(* Step MesCheckResult_1 *)
(* EN: Step structure *)
IF Step_MesCheckResult_1_active THEN
  (* Timeout Check *)
  IF (SYS_TIME - Step_MesCheckResult_1_entry_time) > MesCheckResult_1.T_MAX THEN Step_MesCheckResult_1_timeout := TRUE; END_IF;

  IF Action_MesCheckResult_1_Exec THEN
    "PLCtoMES"."PLC.Unload_Station7DataSaveReq" := TRUE;
    Action_MesCheckResult_1_Done := TRUE;
  END_IF;
END_IF;

(* Step Bypass_1 *)
(* EN: Step structure *)
IF Step_Bypass_1_active THEN
  (* Timeout Check *)
  IF (SYS_TIME - Step_Bypass_1_entry_time) > Bypass_1.T_MAX THEN Step_Bypass_1_timeout := TRUE; END_IF;

  IF Action_Bypass_1_Exec THEN
    Action_Bypass_1_Done := TRUE;
  END_IF;
END_IF;

(* Step ResetMesUnloadRequest_1 *)
(* EN: Step structure *)
IF Step_ResetMesUnloadRequest_1_active THEN
  (* Timeout Check *)
  IF (SYS_TIME - Step_ResetMesUnloadRequest_1_entry_time) > ResetMesUnloadRequest_1.T_MAX THEN Step_ResetMesUnloadRequest_1_timeout := TRUE; END_IF;

  IF Action_ResetMesUnloadRequest_1_Exec THEN
    "PLCtoMES"."PLC.Unload_Station7DataSaveReq" := FALSE;
    "MEStoPLC"."MES.Unload_ResultsStored7OK" := FALSE;
    "MEStoPLC"."MES.Unload_ResultsStored7NG" := FALSE;
    "MEStoPLC"."MES.Unload_ResultsStored7ReqMesDone" := FALSE;
    Action_ResetMesUnloadRequest_1_Done := TRUE;
  END_IF;
END_IF;

(* Step Step314 *)
(* EN: Step structure *)
IF Step_Step314_active THEN
  (* Timeout Check *)
  IF (SYS_TIME - Step_Step314_entry_time) > Step314.T_MAX THEN Step_Step314_timeout := TRUE; END_IF;

  IF Action_Step314_Exec THEN
    Action_Step314_Done := TRUE;
  END_IF;
END_IF;

(* Step MESOverTime *)
(* EN: Step structure *)
IF Step_MESOverTime_active THEN
  (* Timeout Check *)
  IF (SYS_TIME - Step_MESOverTime_entry_time) > MESOverTime.T_MAX THEN Step_MESOverTime_timeout := TRUE; END_IF;

  IF Action_MESOverTime_Exec THEN
    "ST10_DeviceError".MES_Error.CheckInResultOverTime_7 := TRUE;
    Action_MESOverTime_Done := TRUE;
  END_IF;
END_IF;

(* Step ok_1 *)
(* EN: Step structure *)
IF Step_Ok_1_active THEN
  (* Timeout Check *)
  IF (SYS_TIME - Step_Ok_1_entry_time) > Ok_1.T_MAX THEN Step_Ok_1_timeout := TRUE; END_IF;

  IF Action_Ok_1_Exec THEN
    IF "AutoProcessData".B_Press2.PartStatus = 480 THEN
      "AutoProcessData".B_Press2.PartStatus := 499;
    END_IF;
    Action_Ok_1_Done := TRUE;
  END_IF;
END_IF;

(* Step Prepare MES CheckData_1 *)
(* EN: Step structure *)
IF Step_PrepareMESCheckData_1_active THEN
  (* Timeout Check *)
  IF (SYS_TIME - Step_PrepareMESCheckData_1_entry_time) > PrepareMESCheckData_1.T_MAX THEN Step_PrepareMESCheckData_1_timeout := TRUE; END_IF;

  IF Action_PrepareMESCheckData_1_Exec THEN
    Action_PrepareMESCheckData_1_Done := TRUE;
  END_IF;
END_IF;

(* Transition 399: MES Result OK_1 -> MES Check Finish *)
IF Step_MESResultOK_1_active AND ( "AutoProcessData".B_Press2.PartStatus = 499 ) THEN
  Step_MESResultOK_1_active := FALSE;
  Action_MESResultOK_1_Exec := FALSE;

  Step_MESCheckFinish_active := TRUE;
  Step_MESCheckFinish_entry_time := SYS_TIME; (* Reset Timer *)
  Action_MESCheckFinish_Exec := TRUE;

  Trans_Trans321_executed := TRUE;
END_IF;

(* Transition 500: MES Result -> Bypass_1 *)
IF Step_MESResult_active AND ( TRUE ) THEN
  Step_MESResult_active := FALSE;
  Action_MESResult_Exec := FALSE;

  Step_Bypass_1_active := TRUE;
  Step_Bypass_1_entry_time := SYS_TIME; (* Reset Timer *)
  Action_Bypass_1_Exec := TRUE;

  Trans_Trans407_executed := TRUE;
END_IF;

(* Transition 515: MES Check Finish -> RobotPick (Jump) *)
IF Step_MESCheckFinish_active AND ( TRUE ) THEN
  Step_MESCheckFinish_active := FALSE;
  Action_MESCheckFinish_Exec := FALSE;

  Step_RobotPick_active := TRUE;
  Step_RobotPick_entry_time := SYS_TIME; (* Reset Timer *)
  Action_RobotPick_Exec := TRUE;

  Trans_Trans619_executed := TRUE;
END_IF;

(* Transition 308: Prepare MES CheckData_1 -> MesCheckResult_1 *)
IF Step_PrepareMESCheckData_1_active AND ( PrepareMESCheckData_1.T > T#300ms ) THEN
  Step_PrepareMESCheckData_1_active := FALSE;
  Action_PrepareMESCheckData_1_Exec := FALSE;

  Step_MesCheckResult_1_active := TRUE;
  Step_MesCheckResult_1_entry_time := SYS_TIME; (* Reset Timer *)
  Action_MesCheckResult_1_Exec := TRUE;

  Trans_Trans16_executed := TRUE;
END_IF;

(* Transition 315: MesCheckResult_1 -> MESResultOK_1 *)
IF Step_MesCheckResult_1_active AND ( (NOT "MEStoPLC"."MES.Unload_ResultsStored7OK") AND "MEStoPLC"."MES.Unload_ResultsStored7NG" AND "MEStoPLC"."MES.Unload_ResultsStored7ReqMesDone" ) THEN
  Step_MesCheckResult_1_active := FALSE;
  Action_MesCheckResult_1_Exec := FALSE;

  Step_MESResultOK_1_active := TRUE;
  Step_MESResultOK_1_entry_time := SYS_TIME; (* Reset Timer *)
  Action_MESResultOK_1_Exec := TRUE;

  Trans_Trans315_executed := TRUE;
END_IF;

(* Transition 321: Step313 -> CheckFinish_1 *)
IF Step_Step313_active AND ( TRUE ) THEN
  Step_Step313_active := FALSE;
  Action_Step313_Exec := FALSE;

  Step_CheckFinish_1_active := TRUE;
  Step_CheckFinish_1_entry_time := SYS_TIME; (* Reset Timer *)
  Action_CheckFinish_1_Exec := TRUE;

  Trans_Trans319_executed := TRUE; (* Original: Trans321. Typo in XML? *)
END_IF;

(* Transition 322: MesCheckResult_1 -> MESCheckNG_3 *)
IF Step_MesCheckResult_1_active AND ( "AutoProcessData".B_Press2.PartStatus = 452 ) THEN
  Step_MesCheckResult_1_active := FALSE;
  Action_MesCheckResult_1_Exec := FALSE;

  Step_MESCheckNG_3_active := TRUE;
  Step_MESCheckNG_3_entry_time := SYS_TIME; (* Reset Timer *)
  Action_MESCheckNG_3_Exec := TRUE;

  Trans_Trans322_executed := TRUE;
END_IF;

(* Transition 323: MESCheckNG_3 -> MES Result OK_1 *)
IF Step_MESCheckNG_3_active AND ( "MEStoPLC"."MES.Unload_ResultsStored7OK" AND (NOT "MEStoPLC"."MES.Unload_ResultsStored7NG") AND "MEStoPLC"."MES.Unload_ResultsStored7ReqMesDone" AND ("AutoProcessData".B_Press2.PartStatus <> 450) AND ("AutoProcessData".B_Press2.PartStatus <> 455) ) THEN
  Step_MESCheckNG_3_active := FALSE;
  Action_MESCheckNG_3_Exec := FALSE;

  Step_MESResultOK_1_active := TRUE;
  Step_MESResultOK_1_entry_time := SYS_TIME; (* Reset Timer *)
  Action_MESResultOK_1_Exec := TRUE;

  Trans_Trans323_executed := TRUE;
END_IF;

(* Transition 324: MESCheckNG_3 -> Step314 *)
IF Step_MESCheckNG_3_active AND ( (NOT "MEStoPLC"."MES.Load_Station7ReqMesDone") AND (MesCheckResult_1.T > T#10s) ) THEN
  Step_MESCheckNG_3_active := FALSE;
  Action_MESCheckNG_3_Exec := FALSE;

  Step_Step314_active := TRUE;
  Step_Step314_entry_time := SYS_TIME; (* Reset Timer *)
  Action_Step314_Exec := TRUE;

  Trans_Trans324_executed := TRUE;
END_IF;

(* Transition 325: Bypass_1 -> ResetMesUnloadRequest_1 *)
IF Step_Bypass_1_active AND ( (NOT "Station_Sys".Cmd.OnOffLine) ) THEN
  Step_Bypass_1_active := FALSE;
  Action_Bypass_1_Exec := FALSE;

  Step_ResetMesUnloadRequest_1_active := TRUE;
  Step_ResetMesUnloadRequest_1_entry_time := SYS_TIME; (* Reset Timer *)
  Action_ResetMesUnloadRequest_1_Exec := TRUE;

  Trans_Online_1_executed := TRUE; (* Original: Trans325. Typo in XML? *)
END_IF;

(* Transition 326: ResetMesUnloadRequest_1 -> Prepare MES CheckData_1 *)
IF Step_ResetMesUnloadRequest_1_active AND ( NOT "PLCtoMES"."PLC.Unload_Station7DataSaveReq" AND NOT "MEStoPLC"."MES.Unload_ResultsStored7OK" AND NOT "MEStoPLC"."MES.Unload_ResultsStored7NG" AND NOT "MEStoPLC"."MES.Unload_ResultsStored7ReqMesDone" ) THEN
  Step_ResetMesUnloadRequest_1_active := FALSE;
  Action_ResetMesUnloadRequest_1_Exec := FALSE;

  Step_PrepareMESCheckData_1_active := TRUE;
  Step_PrepareMESCheckData_1_entry_time := SYS_TIME; (* Reset Timer *)
  Action_PrepareMESCheckData_1_Exec := TRUE;

  Trans_Trans260_executed := TRUE;
END_IF;

(* Transition 327: Bypass_1 -> ok_1 *)
IF Step_Bypass_1_active AND ( "Station_Sys".Cmd.OnOffLine ) THEN
  Step_Bypass_1_active := FALSE;
  Action_Bypass_1_Exec := FALSE;

  Step_Ok_1_active := TRUE;
  Step_Ok_1_entry_time := SYS_TIME; (* Reset Timer *)
  Action_Ok_1_Exec := TRUE;

  Trans_Trans327_executed := TRUE;
END_IF;

(* Transition 328: MESOverTime -> Bypass_1 (Jump) *)
IF Step_MESOverTime_active AND ( TRUE ) THEN
  Step_MESOverTime_active := FALSE;
  Action_MESOverTime_Exec := FALSE;

  Step_Bypass_1_active := TRUE;
  Step_Bypass_1_entry_time := SYS_TIME; (* Reset Timer *)
  Action_Bypass_1_Exec := TRUE;

  Trans_Trans329_executed := TRUE; (* Original: Trans328. Typo in XML? *)
END_IF;

(* Transition 331: ok_1 -> Step314 *)
IF Step_Ok_1_active AND ( TRUE ) THEN
  Step_Ok_1_active := FALSE;
  Action_Ok_1_Exec := FALSE;

  Step_Step314_active := TRUE;
  Step_Step314_entry_time := SYS_TIME; (* Reset Timer *)
  Action_Step314_Exec := TRUE;

  Trans_Trans328_executed := TRUE; (* Original: Trans331. Typo in XML? *)
END_IF;

(* Transition 330: Step314 -> MESOverTime *)
IF Step_Step314_active AND ( TRUE ) THEN
  Step_Step314_active := FALSE;
  Action_Step314_Exec := FALSE;

  Step_MESOverTime_active := TRUE;
  Step_MESOverTime_entry_time := SYS_TIME; (* Reset Timer *)
  Action_MESOverTime_Exec := TRUE;

  Trans_Trans327_executed := TRUE; (* Original: Trans330. Typo in XML? *)
END_IF;


(* Sequence: S600-S699 RobotPick *)
(* S600-S699工件放行 *)
(* Step RobotPick *)
(* EN: Step structure *)
IF Step_RobotPick_active THEN
  (* Timeout Check *)
  IF (SYS_TIME - Step_RobotPick_entry_time) > RobotPick.T_MAX THEN Step_RobotPick_timeout := TRUE; END_IF;

  IF Action_RobotPick_Exec THEN
    Action_RobotPick_Done := TRUE;
  END_IF;
END_IF;

(* Step ProcessFinsh *)
(* ZH-CN: 正式使用时，需要激活复位空循环 *)
(* EN: Step structure *)
IF Step_ProcessFinsh_3_active THEN
  (* Timeout Check *)
  IF (SYS_TIME - Step_ProcessFinsh_3_entry_time) > ProcessFinsh_3.T_MAX THEN Step_ProcessFinsh_3_timeout := TRUE; END_IF;

  IF Action_ProcessFinsh_3_Exec THEN
    #ioPM_Inface.ProcessComplete := TRUE;
    #ioPM_Inface.ProcessStart := FALSE;
    Action_ProcessFinsh_3_Done := TRUE;
  END_IF;
END_IF;

(* Step DataClear *)
(* EN: Step structure *)
IF Step_DataClear_active THEN
  (* Timeout Check *)
  IF (SYS_TIME - Step_DataClear_entry_time) > DataClear.T_MAX THEN Step_DataClear_timeout := TRUE; END_IF;

  IF Action_DataClear_Exec THEN
    #ioPM_Inface.ProcessResult := 0;
    #ioStatus := 0;
    Action_DataClear_Done := TRUE;
  END_IF;
END_IF;

(* Step Request robot pick *)
(* EN: Step structure *)
IF Step_RequestRobotPick_active THEN
  (* Timeout Check *)
  IF (SYS_TIME - Step_RequestRobotPick_entry_time) > RequestRobotPick.T_MAX THEN Step_RequestRobotPick_timeout := TRUE; END_IF;

  IF Action_RequestRobotPick_Exec THEN
    "AutoProcessControl".B_Press_2.Robot3PickPrimit := TRUE;
    Action_RequestRobotPick_Done := TRUE;
  END_IF;
END_IF;

(* Step Wait robot finish task *)
(* EN: Step structure *)
IF Step_WaitRobotFinishTask_1_active THEN
  (* Timeout Check *)
  IF (SYS_TIME - Step_WaitRobotFinishTask_1_entry_time) > WaitRobotFinishTask_1.T_MAX THEN Step_WaitRobotFinishTask_1_timeout := TRUE; END_IF;

  IF Action_WaitRobotFinishTask_1_Exec THEN
    Action_WaitRobotFinishTask_1_Done := TRUE;
  END_IF;
END_IF;

(* Step DataMove *)
(* EN: Step structure *)
IF Step_DataMove_active THEN
  (* Timeout Check *)
  IF (SYS_TIME - Step_DataMove_entry_time) > DataMove.T_MAX THEN Step_DataMove_timeout := TRUE; END_IF;

  IF Action_DataMove_Exec THEN
    Action_DataMove_Done := TRUE;
  END_IF;
END_IF;

(* Step Wait robot in safety area *)
(* EN: Step structure *)
IF Step_WaitRobotInSafetyArea_active THEN
  (* Timeout Check *)
  IF (SYS_TIME - Step_WaitRobotInSafetyArea_entry_time) > WaitRobotInSafetyArea.T_MAX THEN Step_WaitRobotInSafetyArea_timeout := TRUE; END_IF;

  IF Action_WaitRobotInSafetyArea_Exec THEN
    Action_WaitRobotInSafetyArea_Done := TRUE;
  END_IF;
END_IF;

(* Step PressProgram_1 *)
(* EN: Step structure *)
IF Step_PressProgram_1_active THEN
  (* Timeout Check *)
  IF (SYS_TIME - Step_PressProgram_1_entry_time) > PressProgram_1.T_MAX THEN Step_PressProgram_1_timeout := TRUE; END_IF;

  IF Action_PressProgram_1_Exec THEN
    IF NOT "ST10_GeneralData".FunctionDeSelect.B.FunctionDeSelected_TestPress375A1 THEN
      "DB_maXYmosNC2".ProgNo := 1;
    END_IF;
    Action_PressProgram_1_Done := TRUE;
  END_IF;
END_IF;

(* Step PressHoming_1 *)
(* EN: Step structure *)
IF Step_PressHoming_1_active THEN
  (* Timeout Check *)
  IF (SYS_TIME - Step_PressHoming_1_entry_time) > PressHoming_1.T_MAX THEN Step_PressHoming_1_timeout := TRUE; END_IF;

  IF Action_PressHoming_1_Exec THEN
    "DB_maXYmosNC2".Homing := TRUE;
    Action_PressHoming_1_Done := TRUE;
  END_IF;
END_IF;

(* Step PressReady?_1 *)
(* EN: Step structure *)
IF Step_PressReady_q_1_active THEN
  (* Timeout Check *)
  IF (SYS_TIME - Step_PressReady_q_1_entry_time) > PressReady_q_1.T_MAX THEN Step_PressReady_q_1_timeout := TRUE; END_IF;

  IF Action_PressReady_q_1_Exec THEN
    Action_PressReady_q_1_Done := TRUE;
  END_IF;
END_IF;

(* Step PressHoming?_1 *)
(* EN: Step structure *)
IF Step_PressHoming_q_1_active THEN
  (* Timeout Check *)
  IF (SYS_TIME - Step_PressHoming_q_1_entry_time) > PressHoming_q_1.T_MAX THEN Step_PressHoming_q_1_timeout := TRUE; END_IF;

  IF Action_PressHoming_q_1_Exec THEN
    Action_PressHoming_q_1_Done := TRUE;
  END_IF;
END_IF;

(* Step Step15 *)
(* EN: Step structure *)
IF Step_Step15_active THEN
  (* Timeout Check *)
  IF (SYS_TIME - Step_Step15_entry_time) > Step15.T_MAX THEN Step_Step15_timeout := TRUE; END_IF;

  IF Action_Step15_Exec THEN
    Action_Step15_Done := TRUE;
  END_IF;
END_IF;

(* Step B-PressFitting-01CylinderToHP_1 *)
(* EN: Step structure *)
IF Step_B_PressFitting_01CylinderToHP_1_active THEN
  (* Timeout Check *)
  IF (SYS_TIME - Step_B_PressFitting_01CylinderToHP_1_entry_time) > B_PressFitting_01CylinderToHP_1.T_MAX THEN Step_B_PressFitting_01CylinderToHP_1_timeout := TRUE; END_IF;

  IF Action_B_PressFitting_01CylinderToHP_1_Exec THEN
    "ST10Cylinder".Cy[8].Inout.AutoGoHome := TRUE;
    "ST10Cylinder".Cy[8].Inout.AutoGoWork := FALSE;
    Action_B_PressFitting_01CylinderToHP_1_Done := TRUE;
  END_IF;
END_IF;

(* Transition 600: RobotPick -> PressProgram_1 *)
IF Step_RobotPick_active AND ( TRUE ) THEN
  Step_RobotPick_active := FALSE;
  Action_RobotPick_Exec := FALSE;

  Step_PressProgram_1_active := TRUE;
  Step_PressProgram_1_entry_time := SYS_TIME; (* Reset Timer *)
  Action_PressProgram_1_Exec := TRUE;

  Trans_Trans600_executed := TRUE;
END_IF;

(* Transition 604: DataClear -> ProcessFinsh *)
IF Step_DataClear_active AND ( TRUE ) THEN
  Step_DataClear_active := FALSE;
  Action_DataClear_Exec := FALSE;

  Step_ProcessFinsh_3_active := TRUE;
  Step_ProcessFinsh_3_entry_time := SYS_TIME; (* Reset Timer *)
  Action_ProcessFinsh_3_Exec := TRUE;

  Trans_Trans290_executed := TRUE;
END_IF;

(* Transition 605: ProcessFinsh -> ProcessStart (Jump) *)
IF Step_ProcessFinsh_3_active AND ( TRUE ) THEN
  Step_ProcessFinsh_3_active := FALSE;
  Action_ProcessFinsh_3_Exec := FALSE;

  Step_ProcessStart_active := TRUE;
  Step_ProcessStart_entry_time := SYS_TIME; (* Reset Timer *)
  Action_ProcessStart_Exec := TRUE;

  Trans_Trans699_executed := TRUE;
END_IF;

(* Transition 410: Request robot pick -> Wait robot finish task *)
IF Step_RequestRobotPick_active AND ( "KukaRobot3_CtrlDB".sROBtoPLC.User.Cycle.DO281_PressPickInside AND (NOT "KukaRobot3_CtrlDB".sROBtoPLC.User.Cycle.DO282_PressPickFinish) ) THEN
  Step_RequestRobotPick_active := FALSE;
  Action_RequestRobotPick_Exec := FALSE;

  Step_WaitRobotFinishTask_1_active := TRUE;
  Step_WaitRobotFinishTask_1_entry_time := SYS_TIME; (* Reset Timer *)
  Action_WaitRobotFinishTask_1_Exec := TRUE;

  Trans_Trans412_executed := TRUE;
END_IF;

(* Transition 256: Wait robot finish task -> DataMove *)
IF Step_WaitRobotFinishTask_1_active AND ( "KukaRobot3_CtrlDB".sROBtoPLC.User.Cycle.DO282_PressPickFinish ) THEN
  Step_WaitRobotFinishTask_1_active := FALSE;
  Action_WaitRobotFinishTask_1_Exec := FALSE;

  Step_DataMove_active := TRUE;
  Step_DataMove_entry_time := SYS_TIME; (* Reset Timer *)
  Action_DataMove_Exec := TRUE;

  Trans_Trans257_executed := TRUE;
END_IF;

(* Transition 257: DataMove -> Wait robot in safety area *)
IF Step_DataMove_active AND ( TRUE ) THEN
  Step_DataMove_active := FALSE;
  Action_DataMove_Exec := FALSE;

  Step_WaitRobotInSafetyArea_active := TRUE;
  Step_WaitRobotInSafetyArea_entry_time := SYS_TIME; (* Reset Timer *)
  Action_WaitRobotInSafetyArea_Exec := TRUE;

  Trans_Trans258_executed := TRUE;
END_IF;

(* Transition 258: Wait robot in safety area -> DataClear *)
IF Step_WaitRobotInSafetyArea_active AND ( "KukaRobot3_CtrlDB".sROBtoPLC.User.Home.DO177_PressPut1Area AND "KukaRobot3_CtrlDB".sROBtoPLC.User.Home.DO178_Robot2Area ) THEN
  Step_WaitRobotInSafetyArea_active := FALSE;
  Action_WaitRobotInSafetyArea_Exec := FALSE;

  Step_DataClear_active := TRUE;
  Step_DataClear_entry_time := SYS_TIME; (* Reset Timer *)
  Action_DataClear_Exec := TRUE;

  Trans_Trans261_executed := TRUE;
END_IF;

(* Transition 26: PressHoming_1 -> Step15 *)
IF Step_PressHoming_1_active AND ( "DB_maXYmosNC2".oInHomePos ) THEN
  Step_PressHoming_1_active := FALSE;
  Action_PressHoming_1_Exec := FALSE;

  Step_Step15_active := TRUE;
  Step_Step15_entry_time := SYS_TIME; (* Reset Timer *)
  Action_Step15_Exec := TRUE;

  Trans_Trans9_executed := TRUE; (* Original: Trans26. Typo in XML? *)
END_IF;

(* Transition 27: PressProgram_1 -> PressReady?_1 *)
IF Step_PressProgram_1_active AND ( TRUE ) THEN
  Step_PressProgram_1_active := FALSE;
  Action_PressProgram_1_Exec := FALSE;

  Step_PressReady_q_1_active := TRUE;
  Step_PressReady_q_1_entry_time := SYS_TIME; (* Reset Timer *)
  Action_PressReady_q_1_Exec := TRUE;

  Trans_Trans31_executed := TRUE; (* Original: Trans27. Typo in XML? *)
END_IF;

(* Transition 28: PressReady?_1 -> PressHoming?_1 *)
IF Step_PressReady_q_1_active AND ( "DB_maXYmosNC2".oReady AND "DB_maXYmosNC2".oRdyAmp ) THEN
  Step_PressReady_q_1_active := FALSE;
  Action_PressReady_q_1_Exec := FALSE;

  Step_PressHoming_q_1_active := TRUE;
  Step_PressHoming_q_1_entry_time := SYS_TIME; (* Reset Timer *)
  Action_PressHoming_q_1_Exec := TRUE;

  Trans_Trans32_executed := TRUE; (* Original: Trans28. Typo in XML? *)
END_IF;

(* Transition 29: PressHoming?_1 -> PressHoming_1 *)
IF Step_PressHoming_q_1_active AND ( NOT "DB_maXYmosNC2".oInHomePos ) THEN
  Step_PressHoming_q_1_active := FALSE;
  Action_PressHoming_q_1_Exec := FALSE;

  Step_PressHoming_1_active := TRUE;
  Step_PressHoming_1_entry_time := SYS_TIME; (* Reset Timer *)
  Action_PressHoming_1_Exec := TRUE;

  Trans_Trans33_executed := TRUE; (* Original: Trans29. Typo in XML? *)
END_IF;

(* Transition 30: PressHoming?_1 -> Step15 *)
IF Step_PressHoming_q_1_active AND ( "DB_maXYmosNC2".oInHomePos ) THEN
  Step_PressHoming_q_1_active := FALSE;
  Action_PressHoming_q_1_Exec := FALSE;

  Step_Step15_active := TRUE;
  Step_Step15_entry_time := SYS_TIME; (* Reset Timer *)
  Action_Step15_Exec := TRUE;

  Trans_Trans34_executed := TRUE; (* Original: Trans30. Typo in XML? *)
END_IF;

(* Transition 31: Step15 -> B-PressFitting-01CylinderToHP_1 *)
IF Step_Step15_active AND ( TRUE ) THEN
  Step_Step15_active := FALSE;
  Action_Step15_Exec := FALSE;

  Step_B_PressFitting_01CylinderToHP_1_active := TRUE;
  Step_B_PressFitting_01CylinderToHP_1_entry_time := SYS_TIME; (* Reset Timer *)
  Action_B_PressFitting_01CylinderToHP_1_Exec := TRUE;

  Trans_Trans35_executed := TRUE; (* Original: Trans31. Typo in XML? *)
END_IF;

(* Transition 131: B-PressFitting-01CylinderToHP_1 -> Request robot pick *)
IF Step_B_PressFitting_01CylinderToHP_1_active AND ( (NOT "ST10Cylinder".Cy[8].In.WorkPositionSensor) AND "ST10Cylinder".Cy[8].In.HomePositionSensor ) THEN
  Step_B_PressFitting_01CylinderToHP_1_active := FALSE;
  Action_B_PressFitting_01CylinderToHP_1_Exec := FALSE;

  Step_RequestRobotPick_active := TRUE;
  Step_RequestRobotPick_entry_time := SYS_TIME; (* Reset Timer *)
  Action_RequestRobotPick_Exec := TRUE;

  Trans_Trans768_executed := TRUE;
END_IF;

(* Initial Step *)
IF "RT_DATA".MOP.INIT THEN
  Step_F14_Initial_active := TRUE;
  Step_F14_Initial_entry_time := SYS_TIME;
  Action_F14_Initial_Exec := TRUE;
ELSE
  IF NOT Step_F14_Initial_active THEN
    (* Check for all transitions, and activate the next step if condition met *)
    (* Sequence S01-S99 Initial *)
    IF Step_F14_Initial_active AND Trans_Trans1_executed THEN
      Step_F14_Initial_active := FALSE;
      Action_F14_Initial_Exec := FALSE;

      Step_S2_active := TRUE;
      Step_S2_entry_time := SYS_TIME;
      Action_S2_Exec := TRUE;
    ELSIF Step_S2_active AND Trans_Trans2_executed THEN
      Step_S2_active := FALSE;
      Action_S2_Exec := FALSE;

      Step_S3_active := TRUE;
      Step_S3_entry_time := SYS_TIME;
      Action_S3_Exec := TRUE;
    ELSIF Step_S3_active AND Trans_Trans613_executed THEN
      Step_S3_active := FALSE;
      Action_S3_Exec := FALSE;

      Step_S4_active := TRUE;
      Step_S4_entry_time := SYS_TIME;
      Action_S4_Exec := TRUE;
    ELSIF Step_S4_active AND Trans_Trans3_executed THEN
      Step_S4_active := FALSE;
      Action_S4_Exec := FALSE;

      Step_S5_MESInitial_active := TRUE;
      Step_S5_MESInitial_entry_time := SYS_TIME;
      Action_S5_MESInitial_Exec := TRUE;
    ELSIF Step_S5_MESInitial_active AND Trans_Trans325_executed THEN
      Step_S5_MESInitial_active := FALSE;
      Action_S5_MESInitial_Exec := FALSE;

      Step_CheckPressGripStatus_active := TRUE;
      Step_CheckPressGripStatus_entry_time := SYS_TIME;
      Action_CheckPressGripStatus_Exec := TRUE;
    ELSIF Step_CheckPressGripStatus_active AND Trans_Trans19_executed THEN
      Step_CheckPressGripStatus_active := FALSE;
      Action_CheckPressGripStatus_Exec := FALSE;

      Step_CheckRingExist_active := TRUE;
      Step_CheckRingExist_entry_time := SYS_TIME;
      Action_CheckRingExist_Exec := TRUE;
    ELSIF Step_CheckPressGripStatus_active AND Trans_Trans20_executed THEN
      Step_CheckPressGripStatus_active := FALSE;
      Action_CheckPressGripStatus_Exec := FALSE;

      Step_B_PressFitting_01GripperCylinderToWP_active := TRUE;
      Step_B_PressFitting_01GripperCylinderToWP_entry_time := SYS_TIME;
      Action_B_PressFitting_01GripperCylinderToWP_Exec := TRUE;
    ELSIF Step_CheckPressGripStatus_active AND Trans_Trans119_executed THEN
      Step_CheckPressGripStatus_active := FALSE;
      Action_CheckPressGripStatus_Exec := FALSE;

      Step_StatusAlarm_active := TRUE;
      Step_StatusAlarm_entry_time := SYS_TIME;
      Action_StatusAlarm_Exec := TRUE;
    ELSIF Step_StatusAlarm_active AND Trans_Trans120_executed THEN
      Step_StatusAlarm_active := FALSE;
      Action_StatusAlarm_Exec := FALSE;

      Step_CheckPressGripStatus_active := TRUE;
      Step_CheckPressGripStatus_entry_time := SYS_TIME;
      Action_CheckPressGripStatus_Exec := TRUE;
    ELSIF Step_CheckRingExist_active AND Trans_Trans117_executed THEN
      Step_CheckRingExist_active := FALSE;
      Action_CheckRingExist_Exec := FALSE;

      Step_B_PressFitting_01GripperCylinderToHP_active := TRUE;
      Step_B_PressFitting_01GripperCylinderToHP_entry_time := SYS_TIME;
      Action_B_PressFitting_01GripperCylinderToHP_Exec := TRUE;
    ELSIF Step_B_PressFitting_01GripperCylinderToHP_active AND Trans_Trans765_executed THEN
      Step_B_PressFitting_01GripperCylinderToHP_active := FALSE;
      Action_B_PressFitting_01GripperCylinderToHP_Exec := FALSE;

      Step_PressProgram_active := TRUE;
      Step_PressProgram_entry_time := SYS_TIME;
      Action_PressProgram_Exec := TRUE;
    ELSIF Step_B_PressFitting_01GripperCylinderToWP_active AND Trans_Trans766_executed THEN
      Step_B_PressFitting_01GripperCylinderToWP_active := FALSE;
      Action_B_PressFitting_01GripperCylinderToWP_Exec := FALSE;

      Step_PressProgram_active := TRUE;
      Step_PressProgram_entry_time := SYS_TIME;
      Action_PressProgram_Exec := TRUE;
    ELSIF Step_PressProgram_active AND Trans_Trans10_executed THEN
      Step_PressProgram_active := FALSE;
      Action_PressProgram_Exec := FALSE;

      Step_PressReady_q_active := TRUE;
      Step_PressReady_q_entry_time := SYS_TIME;
      Action_PressReady_q_Exec := TRUE;
    ELSIF Step_PressReady_q_active AND Trans_Trans12_executed THEN
      Step_PressReady_q_active := FALSE;
      Action_PressReady_q_Exec := FALSE;

      Step_PressHoming_q_active := TRUE;
      Step_PressHoming_q_entry_time := SYS_TIME;
      Action_PressHoming_q_Exec := TRUE;
    ELSIF Step_PressHoming_q_active AND Trans_Trans15_executed THEN
      Step_PressHoming_q_active := FALSE;
      Action_PressHoming_q_Exec := FALSE;

      Step_PressHoming_active := TRUE;
      Step_PressHoming_entry_time := SYS_TIME;
      Action_PressHoming_Exec := TRUE;
    ELSIF Step_PressHoming_q_active AND Trans_Trans17_executed THEN
      Step_PressHoming_q_active := FALSE;
      Action_PressHoming_q_Exec := FALSE;

      Step_Step14_active := TRUE;
      Step_Step14_entry_time := SYS_TIME;
      Action_Step14_Exec := TRUE;
    ELSIF Step_PressHoming_active AND Trans_Trans7_executed THEN
      Step_PressHoming_active := FALSE;
      Action_PressHoming_Exec := FALSE;

      Step_Step14_active := TRUE;
      Step_Step14_entry_time := SYS_TIME;
      Action_Step14_Exec := TRUE;
    ELSIF Step_Step14_active AND Trans_Trans18_executed THEN
      Step_Step14_active := FALSE;
      Action_Step14_Exec := FALSE;

      Step_B_PressFitting_01CylinderToHP_active := TRUE;
      Step_B_PressFitting_01CylinderToHP_entry_time := SYS_TIME;
      Action_B_PressFitting_01CylinderToHP_Exec := TRUE;
    ELSIF Step_B_PressFitting_01CylinderToHP_active AND Trans_Trans767_executed THEN
      Step_B_PressFitting_01CylinderToHP_active := FALSE;
      Action_B_PressFitting_01CylinderToHP_Exec := FALSE;

      Step_S10_InitialFinish_active := TRUE;
      Step_S10_InitialFinish_entry_time := SYS_TIME;
      Action_S10_InitialFinish_Exec := TRUE;
    ELSIF Step_S10_InitialFinish_active AND Trans_Trans102_executed THEN
      Step_S10_InitialFinish_active := FALSE;
      Action_S10_InitialFinish_Exec := FALSE;

      Step_ProcessStart_active := TRUE;
      Step_ProcessStart_entry_time := SYS_TIME;
      Action_ProcessStart_Exec := TRUE;

    (* Sequence S100-S199 CheckPartStatus *)
    ELSIF Step_ProcessStart_active AND Trans_Trans200_executed THEN
      Step_ProcessStart_active := FALSE;
      Action_ProcessStart_Exec := FALSE;

      Step_DetermineProductStatus_active := TRUE;
      Step_DetermineProductStatus_entry_time := SYS_TIME;
      Action_DetermineProductStatus_Exec := TRUE;
    ELSIF Step_DetermineProductStatus_active AND Trans_Empty_executed THEN
      Step_DetermineProductStatus_active := FALSE;
      Action_DetermineProductStatus_Exec := FALSE;

      Step_NoPart_active := TRUE;
      Step_NoPart_entry_time := SYS_TIME;
      Action_NoPart_Exec := TRUE;
    ELSIF Step_DetermineProductStatus_active AND Trans_HavePart_executed THEN
      Step_DetermineProductStatus_active := FALSE;
      Action_DetermineProductStatus_Exec := FALSE;

      Step_ShaftOK_active := TRUE;
      Step_ShaftOK_entry_time := SYS_TIME;
      Action_ShaftOK_Exec := TRUE;
    ELSIF Step_DetermineProductStatus_active AND Trans_Trans21_executed THEN
      Step_DetermineProductStatus_active := FALSE;
      Action_DetermineProductStatus_Exec := FALSE;

      Step_ShaftAndRingOK_active := TRUE;
      Step_ShaftAndRingOK_entry_time := SYS_TIME;
      Action_ShaftAndRingOK_Exec := TRUE;
    ELSIF Step_DetermineProductStatus_active AND Trans_Trans22_executed THEN
      Step_DetermineProductStatus_active := FALSE;
      Action_DetermineProductStatus_Exec := FALSE;

      Step_Press_NG_active := TRUE;
      Step_Press_NG_entry_time := SYS_TIME;
      Action_Press_NG_Exec := TRUE;
    ELSIF Step_DetermineProductStatus_active AND Trans_Trans23_executed THEN
      Step_DetermineProductStatus_active := FALSE;
      Action_DetermineProductStatus_Exec := FALSE;

      Step_MES_active := TRUE;
      Step_MES_entry_time := SYS_TIME;
      Action_MES_Exec := TRUE;
    ELSIF Step_DetermineProductStatus_active AND Trans_Trans24_executed THEN
      Step_DetermineProductStatus_active := FALSE;
      Action_DetermineProductStatus_Exec := FALSE;

      Step_MESOK_active := TRUE;
      Step_MESOK_entry_time := SYS_TIME;
      Action_MESOK_Exec := TRUE;
    ELSIF Step_DetermineProductStatus_active AND Trans_Alarm_executed THEN
      Step_DetermineProductStatus_active := FALSE;
      Action_DetermineProductStatus_Exec := FALSE;

      Step_StatusAlarm_1_active := TRUE;
      Step_StatusAlarm_1_entry_time := SYS_TIME;
      Action_StatusAlarm_1_Exec := TRUE;
    ELSIF Step_NoPart_active AND Trans_Trans145_executed THEN
      Step_NoPart_active := FALSE;
      Action_NoPart_Exec := FALSE;

      Step_CheckMachineStatus_active := TRUE;
      Step_CheckMachineStatus_entry_time := SYS_TIME;
      Action_CheckMachineStatus_Exec := TRUE;
    ELSIF Step_ShaftOK_active AND Trans_Trans303_executed THEN
      Step_ShaftOK_active := FALSE;
      Action_ShaftOK_Exec := FALSE;

      Step_PutRing_active := TRUE;
      Step_PutRing_entry_time := SYS_TIME;
      Action_PutRing_Exec := TRUE;
    ELSIF Step_StatusAlarm_1_active AND Trans_Trans304_executed THEN
      Step_StatusAlarm_1_active := FALSE;
      Action_StatusAlarm_1_Exec := FALSE;

      Step_DetermineProductStatus_active := TRUE;
      Step_DetermineProductStatus_entry_time := SYS_TIME;
      Action_DetermineProductStatus_Exec := TRUE;
    ELSIF Step_CheckMachineStatus_active AND Trans_Trans266_executed THEN
      Step_CheckMachineStatus_active := FALSE;
      Action_CheckMachineStatus_Exec := FALSE;

      Step_NormalMode_active := TRUE;
      Step_NormalMode_entry_time := SYS_TIME;
      Action_NormalMode_Exec := TRUE;
    ELSIF Step_NormalMode_active AND Trans_Trans11_executed THEN
      Step_NormalMode_active := FALSE;
      Action_NormalMode_Exec := FALSE;

      Step_ProcessStart_CTStart_active := TRUE;
      Step_ProcessStart_CTStart_entry_time := SYS_TIME;
      Action_ProcessStart_CTStart_Exec := TRUE;
    ELSIF Step_ProcessStart_CTStart_active AND Trans_Trans249_executed THEN
      Step_ProcessStart_CTStart_active := FALSE;
      Action_ProcessStart_CTStart_Exec := FALSE;

      Step_RequestRobotPutShaft_active := TRUE;
      Step_RequestRobotPutShaft_entry_time := SYS_TIME;
      Action_RequestRobotPutShaft_Exec := TRUE;
    ELSIF Step_RequestRobotPutShaft_active AND Trans_Trans283_executed THEN
      Step_RequestRobotPutShaft_active := FALSE;
      Action_RequestRobotPutShaft_Exec := FALSE;

      Step_WaitRobotFinishTask_active := TRUE;
      Step_WaitRobotFinishTask_entry_time := SYS_TIME;
      Action_WaitRobotFinishTask_Exec := TRUE;
    ELSIF Step_PutRing_active AND Trans_Trans125_executed THEN
      Step_PutRing_active := FALSE;
      Action_PutRing_Exec := FALSE;

      Step_RequestRobotPutRing_active := TRUE;
      Step_RequestRobotPutRing_entry_time := SYS_TIME;
      Action_RequestRobotPutRing_Exec := TRUE;
    ELSIF Step_RequestRobotPutRing_active AND Trans_Trans284_executed THEN
      Step_RequestRobotPutRing_active := FALSE;
      Action_RequestRobotPutRing_Exec := FALSE;

      Step_WaitRobotFinishTask_1_1_active := TRUE;
      Step_WaitRobotFinishTask_1_1_entry_time := SYS_TIME;
      Action_WaitRobotFinishTask_1_1_Exec := TRUE;
    ELSIF Step_WaitRobotFinishTask_active AND Trans_Trans146_executed THEN
      Step_WaitRobotFinishTask_active := FALSE;
      Action_WaitRobotFinishTask_Exec := FALSE;

      Step_RobotLeavePress_Area_active := TRUE;
      Step_RobotLeavePress_Area_entry_time := SYS_TIME;
      Action_RobotLeavePress_Area_Exec := TRUE;
    ELSIF Step_WaitRobotFinishTask_1_1_active AND Trans_Trans147_executed THEN
      Step_WaitRobotFinishTask_1_1_active := FALSE;
      Action_WaitRobotFinishTask_1_1_Exec := FALSE;

      Step_PartStatus_active := TRUE;
      Step_PartStatus_entry_time := SYS_TIME;
      Action_PartStatus_Exec := TRUE;
    ELSIF Step_RobotLeavePress_Area_active AND Trans_Trans199_executed THEN
      Step_RobotLeavePress_Area_active := FALSE;
      Action_RobotLeavePress_Area_Exec := FALSE;

      Step_PartCheck_active := TRUE;
      Step_PartCheck_entry_time := SYS_TIME;
      Action_PartCheck_Exec := TRUE;
    ELSIF Step_PartStatus_active AND Trans_Trans124_executed THEN
      Step_PartStatus_active := FALSE;
      Action_PartStatus_Exec := FALSE;

      Step_RobotLeavePressArea_1_active := TRUE;
      Step_RobotLeavePressArea_1_entry_time := SYS_TIME;
      Action_RobotLeavePressArea_1_Exec := TRUE;
    ELSIF Step_RobotLeavePressArea_1_active AND Trans_Trans236_executed THEN
      Step_RobotLeavePressArea_1_active := FALSE;
      Action_RobotLeavePressArea_1_Exec := FALSE;

      Step_Part_Check_active := TRUE;
      Step_Part_Check_entry_time := SYS_TIME;
      Action_Part_Check_Exec := TRUE;
    ELSIF Step_PartCheck_active AND Trans_Trans252_executed THEN
      Step_PartCheck_active := FALSE;
      Action_PartCheck_Exec := FALSE;

      Step_PutRing_active := TRUE;
      Step_PutRing_entry_time := SYS_TIME;
      Action_PutRing_Exec := TRUE;
    ELSIF Step_PartCheck_active AND Trans_Trans263_executed THEN
      Step_PartCheck_active := FALSE;
      Action_PartCheck_Exec := FALSE;

      Step_ProductCheckAlarm_active := TRUE;
      Step_ProductCheckAlarm_entry_time := SYS_TIME;
      Action_ProductCheckAlarm_Exec := TRUE;
    ELSIF Step_Part_Check_active AND Trans_Trans262_executed THEN
      Step_Part_Check_active := FALSE;
      Action_Part_Check_Exec := FALSE;

      Step_ProcessFInish_2_active := TRUE;
      Step_ProcessFInish_2_entry_time := SYS_TIME;
      Action_ProcessFInish_2_Exec := TRUE;
    ELSIF Step_Part_Check_active AND Trans_Trans267_executed THEN
      Step_Part_Check_active := FALSE;
      Action_Part_Check_Exec := FALSE;

      Step_ProductCheckAlarm_1_active := TRUE;
      Step_ProductCheckAlarm_1_entry_time := SYS_TIME;
      Action_ProductCheckAlarm_1_Exec := TRUE;
    ELSIF Step_ProductCheckAlarm_active AND Trans_Trans265_executed THEN
      Step_ProductCheckAlarm_active := FALSE;
      Action_ProductCheckAlarm_Exec := FALSE;

      Step_PartCheck_active := TRUE;
      Step_PartCheck_entry_time := SYS_TIME;
      Action_PartCheck_Exec := TRUE;
    ELSIF Step_ProductCheckAlarm_1_active AND Trans_Trans269_executed THEN
      Step_ProductCheckAlarm_1_active := FALSE;
      Action_ProductCheckAlarm_1_Exec := FALSE;

      Step_Part_Check_active := TRUE;
      Step_Part_Check_entry_time := SYS_TIME;
      Action_Part_Check_Exec := TRUE;
    ELSIF Step_PartStatus_active AND Trans_Trans138_executed THEN
      Step_PartStatus_active := FALSE;
      Action_PartStatus_Exec := FALSE;

      Step_MES_1NG_active := TRUE;
      Step_MES_1NG_entry_time := SYS_TIME;
      Action_MES_1NG_Exec := TRUE;
    ELSIF Step_MES_1NG_active AND Trans_Trans36_executed THEN
      Step_MES_1NG_active := FALSE;
      Action_MES_1NG_Exec := FALSE;

      Step_RobotPick_active := TRUE;
      Step_RobotPick_entry_time := SYS_TIME;
      Action_RobotPick_Exec := TRUE;
    ELSIF Step_ShaftAndRingOK_active AND Trans_Trans21_executed THEN
      Step_ShaftAndRingOK_active := FALSE;
      Action_ShaftAndRingOK_Exec := FALSE;

      Step_ProcessFInish_2_active := TRUE;
      Step_ProcessFInish_2_entry_time := SYS_TIME;
      Action_ProcessFInish_2_Exec := TRUE;
    ELSIF Step_Press_NG_active AND Trans_Trans22_executed THEN
      Step_Press_NG_active := FALSE;
      Action_Press_NG_Exec := FALSE;

      Step_ProcessFInish_1_active := TRUE;
      Step_ProcessFInish_1_entry_time := SYS_TIME;
      Action_ProcessFInish_1_Exec := TRUE;
    ELSIF Step_MES_active AND Trans_Trans23_executed THEN
      Step_MES_active := FALSE;
      Action_MES_Exec := FALSE;

      Step_ProcessFInish_1_active := TRUE;
      Step_ProcessFInish_1_entry_time := SYS_TIME;
      Action_ProcessFInish_1_Exec := TRUE;
    ELSIF Step_MESOK_active AND Trans_Trans25_executed THEN
      Step_MESOK_active := FALSE;
      Action_MESOK_Exec := FALSE;

      Step_RobotPick_active := TRUE;
      Step_RobotPick_entry_time := SYS_TIME;
      Action_RobotPick_Exec := TRUE;
    ELSIF Step_ProcessFInish_2_active AND Trans_Trans250_executed THEN
      Step_ProcessFInish_2_active := FALSE;
      Action_ProcessFInish_2_Exec := FALSE;

      Step_MES_Check_In_active := TRUE;
      Step_MES_Check_In_entry_time := SYS_TIME;
      Action_MES_Check_In_Exec := TRUE;

    (* Sequence S150-S199 MES Check In *)
    ELSIF Step_MES_Check_In_active AND Trans_Trans139_executed THEN
      Step_MES_Check_In_active := FALSE;
      Action_MES_Check_In_Exec := FALSE;

      Step_Bypass_active := TRUE;
      Step_Bypass_entry_time := SYS_TIME;
      Action_Bypass_Exec := TRUE;
    ELSIF Step_Bypass_active AND Trans_Trans317_executed THEN
      Step_Bypass_active := FALSE;
      Action_Bypass_Exec := FALSE;

      Step_Bypass_1_active := TRUE;
      Step_Bypass_1_entry_time := SYS_TIME;
      Action_Bypass_1_Exec := TRUE;
    ELSIF Step_Bypass_active AND Trans_Online_executed THEN
      Step_Bypass_active := FALSE;
      Action_Bypass_Exec := FALSE;

      Step_ResetMesCheckRequest_active := TRUE;
      Step_ResetMesCheckRequest_entry_time := SYS_TIME;
      Action_ResetMesCheckRequest_Exec := TRUE;
    ELSIF Step_ResetMesCheckRequest_active AND Trans_Trans318_executed THEN
      Step_ResetMesCheckRequest_active := FALSE;
      Action_ResetMesCheckRequest_Exec := FALSE;

      Step_ResetMesCheckRequest_active := TRUE;
      Step_ResetMesCheckRequest_entry_time := SYS_TIME;
      Action_ResetMesCheckRequest_Exec := TRUE;
    ELSIF Step_ResetMesCheckRequest_active AND Trans_Trans259_executed THEN
      Step_ResetMesCheckRequest_active := FALSE;
      Action_ResetMesCheckRequest_Exec := FALSE;

      Step_PrepareMESCheckData_active := TRUE;
      Step_PrepareMESCheckData_entry_time := SYS_TIME;
      Action_PrepareMESCheckData_Exec := TRUE;
    ELSIF Step_PrepareMESCheckData_active AND Trans_Trans26_executed THEN
      Step_PrepareMESCheckData_active := FALSE;
      Action_PrepareMESCheckData_Exec := FALSE;

      Step_MesCheckIn_1_active := TRUE;
      Step_MesCheckIn_1_entry_time := SYS_TIME;
      Action_MesCheckIn_1_Exec := TRUE;
    ELSIF Step_MesCheckIn_1_active AND Trans_Trans313_executed THEN
      Step_MesCheckIn_1_active := FALSE;
      Action_MesCheckIn_1_Exec := FALSE;

      Step_Step313_active := TRUE;
      Step_Step313_entry_time := SYS_TIME;
      Action_Step313_Exec := TRUE;
    ELSIF Step_MesCheckIn_1_active AND Trans_Trans316_executed THEN
      Step_MesCheckIn_1_active := FALSE;
      Action_MesCheckIn_1_Exec := FALSE;

      Step_MESCheckNG_2_active := TRUE;
      Step_MESCheckNG_2_entry_time := SYS_TIME;
      Action_MESCheckNG_2_Exec := TRUE;
    ELSIF Step_MesCheckIn_1_active AND Trans_Trans302_executed THEN
      Step_MesCheckIn_1_active := FALSE;
      Action_MesCheckIn_1_Exec := FALSE;

      Step_MESOverTime_1_active := TRUE;
      Step_MESOverTime_1_entry_time := SYS_TIME;
      Action_MESOverTime_1_Exec := TRUE;
    ELSIF Step_Step313_active AND Trans_Trans319_executed THEN
      Step_Step313_active := FALSE;
      Action_Step313_Exec := FALSE;

      Step_CheckFinish_1_active := TRUE;
      Step_CheckFinish_1_entry_time := SYS_TIME;
      Action_CheckFinish_1_Exec := TRUE;
    ELSIF Step_MESCheckNG_2_active AND Trans_Trans315_executed THEN
      Step_MESCheckNG_2_active := FALSE;
      Action_MESCheckNG_2_Exec := FALSE;

      Step_CheckFinish_1_active := TRUE;
      Step_CheckFinish_1_entry_time := SYS_TIME;
      Action_CheckFinish_1_Exec := TRUE;
    ELSIF Step_MESOverTime_1_active AND Trans_Trans320_executed THEN
      Step_MESOverTime_1_active := FALSE;
      Action_MESOverTime_1_Exec := FALSE;

      Step_Bypass_active := TRUE;
      Step_Bypass_entry_time := SYS_TIME;
      Action_Bypass_Exec := TRUE;
    ELSIF Step_CheckFinish_1_active AND Trans_Trans311_executed THEN
      Step_CheckFinish_1_active := FALSE;
      Action_CheckFinish_1_Exec := FALSE;

      Step_Pressing_active := TRUE;
      Step_Pressing_entry_time := SYS_TIME;
      Action_Pressing_Exec := TRUE;

    (* Sequence S200-S299Pressing *)
    ELSIF Step_Pressing_active AND Trans_Trans147_executed THEN
      Step_Pressing_active := FALSE;
      Action_Pressing_Exec := FALSE;

      Step_CheckPressReady_active := TRUE;
      Step_CheckPressReady_entry_time := SYS_TIME;
      Action_CheckPressReady_Exec := TRUE;
    ELSIF Step_CheckPressReady_active AND Trans_Trans211_executed THEN
      Step_CheckPressReady_active := FALSE;
      Action_CheckPressReady_Exec := FALSE;

      Step_CheckPressProgram_active := TRUE;
      Step_CheckPressProgram_entry_time := SYS_TIME;
      Action_CheckPressProgram_Exec := TRUE;
    ELSIF Step_CheckPressProgram_active AND Trans_Trans130_executed THEN
      Step_CheckPressProgram_active := FALSE;
      Action_CheckPressProgram_Exec := FALSE;

      Step_StartCycle_active := TRUE;
      Step_StartCycle_entry_time := SYS_TIME;
      Action_StartCycle_Exec := TRUE;
    ELSIF Step_StartCycle_active AND Trans_Trans132_executed THEN
      Step_StartCycle_active := FALSE;
      Action_StartCycle_Exec := FALSE;

      Step_CheckPressSensor_active := TRUE;
      Step_CheckPressSensor_entry_time := SYS_TIME;
      Action_CheckPressSensor_Exec := TRUE;
    ELSIF Step_CheckPressSensor_active AND Trans_Trans129_executed THEN
      Step_CheckPressSensor_active := FALSE;
      Action_CheckPressSensor_Exec := FALSE;

      Step_PartStatus_1_active := TRUE;
      Step_PartStatus_1_entry_time := SYS_TIME;
      Action_PartStatus_1_Exec := TRUE;
    ELSIF Step_PartStatus_1_active AND Trans_Trans128_executed THEN
      Step_PartStatus_1_active := FALSE;
      Action_PartStatus_1_Exec := FALSE;

      Step_WaitPressFinish_active := TRUE;
      Step_WaitPressFinish_entry_time := SYS_TIME;
      Action_WaitPressFinish_Exec := TRUE;
    ELSIF Step_WaitPressFinish_active AND Trans_Trans201_executed THEN
      Step_WaitPressFinish_active := FALSE;
      Action_WaitPressFinish_Exec := FALSE;

      Step_ResetPressStart_active := TRUE;
      Step_ResetPressStart_entry_time := SYS_TIME;
      Action_ResetPressStart_Exec := TRUE;
    ELSIF Step_ResetPressStart_active AND Trans_Trans133_executed THEN
      Step_ResetPressStart_active := FALSE;
      Action_ResetPressStart_Exec := FALSE;

      Step_CheckPressResult_active := TRUE;
      Step_CheckPressResult_entry_time := SYS_TIME;
      Action_CheckPressResult_Exec := TRUE;
    ELSIF Step_CheckPressResult_active AND Trans_Trans135_executed THEN
      Step_CheckPressResult_active := FALSE;
      Action_CheckPressResult_Exec := FALSE;

      Step_ResultOKData_active := TRUE;
      Step_ResultOKData_entry_time := SYS_TIME;
      Action_ResultOKData_Exec := TRUE;
    ELSIF Step_CheckPressResult_active AND Trans_Trans142_executed THEN
      Step_CheckPressResult_active := FALSE;
      Action_CheckPressResult_Exec := FALSE;

      Step_ResultNGData_active := TRUE;
      Step_ResultNGData_entry_time := SYS_TIME;
      Action_ResultNGData_Exec := TRUE;
    ELSIF Step_ResultOKData_active AND Trans_Trans136_executed THEN
      Step_ResultOKData_active := FALSE;
      Action_ResultOKData_Exec := FALSE;

      Step_Step147_active := TRUE;
      Step_Step147_entry_time := SYS_TIME;
      Action_Step147_Exec := TRUE;
    ELSIF Step_ResultNGData_active AND Trans_Trans143_executed THEN
      Step_ResultNGData_active := FALSE;
      Action_ResultNGData_Exec := FALSE;

      Step_Step147_active := TRUE;
      Step_Step147_entry_time := SYS_TIME;
      Action_Step147_Exec := TRUE;
    ELSIF Step_Step147_active AND Trans_Trans144_executed THEN
      Step_Step147_active := FALSE;
      Action_Step147_Exec := FALSE;

      Step_ProcessFInish_1_active := TRUE;
      Step_ProcessFInish_1_entry_time := SYS_TIME;
      Action_ProcessFInish_1_Exec := TRUE;
    ELSIF Step_ProcessFInish_1_active AND Trans_Trans134_executed THEN
      Step_ProcessFInish_1_active := FALSE;
      Action_ProcessFInish_1_Exec := FALSE;

      Step_Step400_active := TRUE;
      Step_Step400_entry_time := SYS_TIME;
      Action_Step400_Exec := TRUE;

    (* Sequence S400-S499OK&NG Status Count *)
    ELSIF Step_Step400_active AND Trans_Trans224_executed THEN
      Step_Step400_active := FALSE;
      Action_Step400_Exec := FALSE;

      Step_JudgeStatus_active := TRUE;
      Step_JudgeStatus_entry_time := SYS_TIME;
      Action_JudgeStatus_Exec := TRUE;
    ELSIF Step_JudgeStatus_active AND Trans_OK_executed THEN
      Step_JudgeStatus_active := FALSE;
      Action_JudgeStatus_Exec := FALSE;

      Step_OKCount_active := TRUE;
      Step_OKCount_entry_time := SYS_TIME;
      Action_OKCount_Exec := TRUE;
    ELSIF Step_JudgeStatus_active AND Trans_NG_executed THEN
      Step_JudgeStatus_active := FALSE;
      Action_JudgeStatus_Exec := FALSE;

      Step_NGCount_active := TRUE;
      Step_NGCount_entry_time := SYS_TIME;
      Action_NGCount_Exec := TRUE;
    ELSIF Step_OKCount_active AND Trans_Trans403_executed THEN
      Step_OKCount_active := FALSE;
      Action_OKCount_Exec := FALSE;

      Step_ProcessFinish_active := TRUE;
      Step_ProcessFinish_entry_time := SYS_TIME;
      Action_ProcessFinish_Exec := TRUE;
    ELSIF Step_NGCount_active AND Trans_Trans404_executed THEN
      Step_NGCount_active := FALSE;
      Action_NGCount_Exec := FALSE;

      Step_ProcessFinish_active := TRUE;
      Step_ProcessFinish_entry_time := SYS_TIME;
      Action_ProcessFinish_Exec := TRUE;
    ELSIF Step_ProcessFinish_active AND Trans_Trans405_executed THEN
      Step_ProcessFinish_active := FALSE;
      Action_ProcessFinish_Exec := FALSE;

      Step_MESResult_active := TRUE;
      Step_MESResult_entry_time := SYS_TIME;
      Action_MESResult_Exec := TRUE;

    (* Sequence S500-S599 MES Result *)
    ELSIF Step_MESResult_active AND Trans_Trans407_executed THEN
      Step_MESResult_active := FALSE;
      Action_MESResult_Exec := FALSE;

      Step_Bypass_1_active := TRUE;
      Step_Bypass_1_entry_time := SYS_TIME;
      Action_Bypass_1_Exec := TRUE;
    ELSIF Step_Bypass_1_active AND Trans_Online_1_executed THEN
      Step_Bypass_1_active := FALSE;
      Action_Bypass_1_Exec := FALSE;

      Step_ResetMesUnloadRequest_1_active := TRUE;
      Step_ResetMesUnloadRequest_1_entry_time := SYS_TIME;
      Action_ResetMesUnloadRequest_1_Exec := TRUE;
    ELSIF Step_Bypass_1_active AND Trans_Trans327_executed THEN
      Step_Bypass_1_active := FALSE;
      Action_Bypass_1_Exec := FALSE;

      Step_Ok_1_active := TRUE;
      Step_Ok_1_entry_time := SYS_TIME;
      Action_Ok_1_Exec := TRUE;
    ELSIF Step_ResetMesUnloadRequest_1_active AND Trans_Trans260_executed THEN
      Step_ResetMesUnloadRequest_1_active := FALSE;
      Action_ResetMesUnloadRequest_1_Exec := FALSE;

      Step_PrepareMESCheckData_1_active := TRUE;
      Step_PrepareMESCheckData_1_entry_time := SYS_TIME;
      Action_PrepareMESCheckData_1_Exec := TRUE;
    ELSIF Step_Ok_1_active AND Trans_Trans328_executed THEN
      Step_Ok_1_active := FALSE;
      Action_Ok_1_Exec := FALSE;

      Step_Step314_active := TRUE;
      Step_Step314_entry_time := SYS_TIME;
      Action_Step314_Exec := TRUE;
    ELSIF Step_PrepareMESCheckData_1_active AND Trans_Trans16_executed THEN
      Step_PrepareMESCheckData_1_active := FALSE;
      Action_PrepareMESCheckData_1_Exec := FALSE;

      Step_MesCheckResult_1_active := TRUE;
      Step_MesCheckResult_1_entry_time := SYS_TIME;
      Action_MesCheckResult_1_Exec := TRUE;
    ELSIF Step_Step314_active AND Trans_Trans327_executed THEN
      Step_Step314_active := FALSE;
      Action_Step314_Exec := FALSE;

      Step_MESOverTime_active := TRUE;
      Step_MESOverTime_entry_time := SYS_TIME;
      Action_MESOverTime_Exec := TRUE;
    ELSIF Step_MESOverTime_active AND Trans_Trans328_executed THEN
      Step_MESOverTime_active := FALSE;
      Action_MESOverTime_Exec := FALSE;

      Step_Bypass_1_active := TRUE;
      Step_Bypass_1_entry_time := SYS_TIME;
      Action_Bypass_1_Exec := TRUE;
    ELSIF Step_MesCheckResult_1_active AND Trans_Trans315_executed THEN
      Step_MesCheckResult_1_active := FALSE;
      Action_MesCheckResult_1_Exec := FALSE;

      Step_MESResultOK_1_active := TRUE;
      Step_MESResultOK_1_entry_time := SYS_TIME;
      Action_MESResultOK_1_Exec := TRUE;
    ELSIF Step_MesCheckResult_1_active AND Trans_Trans138_executed THEN
      Step_MesCheckResult_1_active := FALSE;
      Action_MesCheckResult_1_Exec := FALSE;

      Step_MESCheckNG_3_active := TRUE;
      Step_MESCheckNG_3_entry_time := SYS_TIME;
      Action_MESCheckNG_3_Exec := TRUE;
    ELSIF Step_MESResultOK_1_active AND Trans_Trans321_executed THEN
      Step_MESResultOK_1_active := FALSE;
      Action_MESResultOK_1_Exec := FALSE;

      Step_MESCheckFinish_active := TRUE;
      Step_MESCheckFinish_entry_time := SYS_TIME;
      Action_MESCheckFinish_Exec := TRUE;
    ELSIF Step_MESCheckNG_3_active AND Trans_Trans322_executed THEN
      Step_MESCheckNG_3_active := FALSE;
      Action_MESCheckNG_3_Exec := FALSE;

      Step_MESResultOK_1_active := TRUE;
      Step_MESResultOK_1_entry_time := SYS_TIME;
      Action_MESResultOK_1_Exec := TRUE;
    ELSIF Step_MESCheckNG_3_active AND Trans_Trans324_executed THEN
      Step_MESCheckNG_3_active := FALSE;
      Action_MESCheckNG_3_Exec := FALSE;

      Step_Step314_active := TRUE;
      Step_Step314_entry_time := SYS_TIME;
      Action_Step314_Exec := TRUE;
    ELSIF Step_MESCheckFinish_active AND Trans_Trans619_executed THEN
      Step_MESCheckFinish_active := FALSE;
      Action_MESCheckFinish_Exec := FALSE;

      Step_RobotPick_active := TRUE;
      Step_RobotPick_entry_time := SYS_TIME;
      Action_RobotPick_Exec := TRUE;

    (* Sequence S600-S699 RobotPick *)
    ELSIF Step_RobotPick_active AND Trans_Trans600_executed THEN
      Step_RobotPick_active := FALSE;
      Action_RobotPick_Exec := FALSE;

      Step_PressProgram_1_active := TRUE;
      Step_PressProgram_1_entry_time := SYS_TIME;
      Action_PressProgram_1_Exec := TRUE;
    ELSIF Step_PressProgram_1_active AND Trans_Trans31_executed THEN
      Step_PressProgram_1_active := FALSE;
      Action_PressProgram_1_Exec := FALSE;

      Step_PressReady_q_1_active := TRUE;
      Step_PressReady_q_1_entry_time := SYS_TIME;
      Action_PressReady_q_1_Exec := TRUE;
    ELSIF Step_PressReady_q_1_active AND Trans_Trans32_executed THEN
      Step_PressReady_q_1_active := FALSE;
      Action_PressReady_q_1_Exec := FALSE;

      Step_PressHoming_q_1_active := TRUE;
      Step_PressHoming_q_1_entry_time := SYS_TIME;
      Action_PressHoming_q_1_Exec := TRUE;
    ELSIF Step_PressHoming_q_1_active AND Trans_Trans33_executed THEN
      Step_PressHoming_q_1_active := FALSE;
      Action_PressHoming_q_1_Exec := FALSE;

      Step_PressHoming_1_active := TRUE;
      Step_PressHoming_1_entry_time := SYS_TIME;
      Action_PressHoming_1_Exec := TRUE;
    ELSIF Step_PressHoming_q_1_active AND Trans_Trans34_executed THEN
      Step_PressHoming_q_1_active := FALSE;
      Action_PressHoming_q_1_Exec := FALSE;

      Step_Step15_active := TRUE;
      Step_Step15_entry_time := SYS_TIME;
      Action_Step15_Exec := TRUE;
    ELSIF Step_PressHoming_1_active AND Trans_Trans9_executed THEN
      Step_PressHoming_1_active := FALSE;
      Action_PressHoming_1_Exec := FALSE;

      Step_Step15_active := TRUE;
      Step_Step15_entry_time := SYS_TIME;
      Action_Step15_Exec := TRUE;
    ELSIF Step_Step15_active AND Trans_Trans35_executed THEN
      Step_Step15_active := FALSE;
      Action_Step15_Exec := FALSE;

      Step_B_PressFitting_01CylinderToHP_1_active := TRUE;
      Step_B_PressFitting_01CylinderToHP_1_entry_time := SYS_TIME;
      Action_B_PressFitting_01CylinderToHP_1_Exec := TRUE;
    ELSIF Step_B_PressFitting_01CylinderToHP_1_active AND Trans_Trans768_executed THEN
      Step_B_PressFitting_01CylinderToHP_1_active := FALSE;
      Action_B_PressFitting_01CylinderToHP_1_Exec := FALSE;

      Step_RequestRobotPick_active := TRUE;
      Step_RequestRobotPick_entry_time := SYS_TIME;
      Action_RequestRobotPick_Exec := TRUE;
    ELSIF Step_RequestRobotPick_active AND Trans_Trans412_executed THEN
      Step_RequestRobotPick_active := FALSE;
      Action_RequestRobotPick_Exec := FALSE;

      Step_WaitRobotFinishTask_1_active := TRUE;
      Step_WaitRobotFinishTask_1_entry_time := SYS_TIME;
      Action_WaitRobotFinishTask_1_Exec := TRUE;
    ELSIF Step_WaitRobotFinishTask_1_active AND Trans_Trans257_executed THEN
      Step_WaitRobotFinishTask_1_active := FALSE;
      Action_WaitRobotFinishTask_1_Exec := FALSE;

      Step_DataMove_active := TRUE;
      Step_DataMove_entry_time := SYS_TIME;
      Action_DataMove_Exec := TRUE;
    ELSIF Step_DataMove_active AND Trans_Trans258_executed THEN
      Step_DataMove_active := FALSE;
      Action_DataMove_Exec := FALSE;

      Step_WaitRobotInSafetyArea_active := TRUE;
      Step_WaitRobotInSafetyArea_entry_time := SYS_TIME;
      Action_WaitRobotInSafetyArea_Exec := TRUE;
    ELSIF Step_WaitRobotInSafetyArea_active AND Trans_Trans261_executed THEN
      Step_WaitRobotInSafetyArea_active := FALSE;
      Action_WaitRobotInSafetyArea_Exec := FALSE;

      Step_DataClear_active := TRUE;
      Step_DataClear_entry_time := SYS_TIME;
      Action_DataClear_Exec := TRUE;
    ELSIF Step_DataClear_active AND Trans_Trans290_executed THEN
      Step_DataClear_active := FALSE;
      Action_DataClear_Exec := FALSE;

      Step_ProcessFinsh_3_active := TRUE;
      Step_ProcessFinsh_3_entry_time := SYS_TIME;
      Action_ProcessFinsh_3_Exec := TRUE;
    END_IF;
  END_IF;
END_IF;


(* Post-Operations *)

(* Network 1 *)
#ioPM_Inface.StepNum := #RT_DATA.S_DISPLAY;

(* Network 2 *)
IF iSysInface.Reset THEN
  #AlarmID := 0;
END_IF;

(* Network 3 *)
TON[10].IN := #工件放行中;
TON[10].PT := T#0.5s;
#工件放行中 := FALSE;

END_FUNCTION_BLOCK